(* CoDeSys 2.3.9.35 project: Program stor plattform.pro *)
(* Libraries: Standard.lib 2.12.10 13:48:34, Iecsfc.lib 2.12.10 13:48:34, SYSLIBCALLBACK.LIB 2.12.10 13:48:34 *)

(* PLC configuration (modules and I/O channels)
K-Bus [K_Bus] node 0, in %IB0 out %QB0
DIN1 AT %IX2300.0 [BOOLOnX_I] Internal Digital Input Bit 1
DIN2 AT %IX2300.1 [BOOLOnX_I] Internal Digital Input Bit 2
DOUT1 AT %QX2300.0 [BOOLOnX_Q] Internal Digital Output Bit 1
DOUT2 AT %QX2300.1 [BOOLOnX_Q] Internal Digital Output Bit 2
Fieldbus variables [FB_VARS] node 3, in %IB0 out %QB0
Flag variables [FLAG_VARS] node 4, in %IB0 out %QB0
*)

(* Task configuration *)
TASK NewTask (PRIORITY := 15); (* freewheeling *)
	PLC_PRG();
	Read_Pos();
	Read_Param();
	SET_STEP();
END_TASK

(* Global variable list: Global_Variables *)
VAR_GLOBAL
	(*Manual mode variabler*)
	STOP: BOOL;
	JOGM1: BOOL;
	JOGP1: BOOL;
	JOGM2: BOOL;
	JOGP2: BOOL;
	JOGM3: BOOL;
	JOGP3: BOOL;
	GO_UP: BOOL;
	GO_DOWN: BOOL;
	GO_HOME: BOOL;
	Manual_speed: INT:=300;

	(*Motor 1*)
	M1_Cont_inhibit AT%QX2404.8 : BOOL;
	DATA_IN_M1: INT;
	Y_M1: INT;
	M1_ANGLE: REAL;

	(*Motor 2*)
	M2_Cont_inhibit AT%QX2411.8 : BOOL;
	DATA_IN_M2: INT;
	Y_M2: INT;
	M2_ANGLE:REAL;

	(*Motor 3*)
	M3_Cont_inhibit AT%QX2418.8 : BOOL;
	DATA_IN_M3: INT;
	Y_M3: INT;
	M3_ANGLE:REAL;




   (*MOTOR 1 Set Points*)
	p1_step: INT;
	(*MOTOR 2 Set Points*)
	p2_step: INT;
	(*MOTOR 3 Set points*)
	p3_step: INT;


	(*Platform angle Set Points*)
	pitch:REAL;
	roll:REAL;


	(*MODES*)
	ENABLE: BOOL;  (*Enables the Drives*)
	manual_run: BOOL;		(* Set specified position *)
	wave_run: BOOL; 	(* Wave PROGRAM *)
	input_run: BOOL;		(* Roll / Pitch input from other sources *)

	SIMULATION_UDP: BOOL;

	LOGG :BOOL;

END_VAR

VAR_GLOBAL CONSTANT

	l1:INT:=150;  			(*lower arm in mm*)
	l2:INT:=330;  			(*upper arm in mm*)
	l3:INT:=1075; 			(*length between joints p1, p2, p3*)
	l4:INT:=931;			(*length of platform center from p1*)
	l5:INT := 311;
	l6:INT := 620;
	mid_length:INT:=370;	(*mid length of both arms combined*)
	min_angle:INT:= -125;
	max_angle:INT:= 0;
	max_roll:INT:=10;
	min_roll:INT:=-10;
	max_pitch:INT:=10;
	min_pitch: INT:=-10;
	am:REAL:=57.2958; 			(*arcminute constant*)

END_VAR

(* POU PLC_PRG, ST *)
PROGRAM PLC_PRG
VAR
	RPTS: ROLL_PITCH_TO_STEP;
	Read_par: BOOL;

END_VAR
(* PROGRAM VELGER. *)

IF(wave_run) AND NOT(input_run) AND NOT(manual_run) THEN
WAVE_V3();
END_IF;

IF(input_run) AND NOT(wave_run) AND NOT(manual_run) THEN
INPUT_MODE();
END_IF;

IF(manual_run) AND NOT(input_run) AND NOT(wave_run) THEN
MANUAL();
END_IF;

(*Setter Plattformen i 0 pos.*)
IF( NOT wave_run AND NOT input_run AND NOT manual_run) THEN
RPTS(roll_angle:=0,pitch_angle:=0);
p1_step:=RPTS.step1;
p2_step:=RPTS.step2;
p3_step:=RPTS.step3;
END_IF;
END_PROGRAM

(* POU Calculations/ROLL_PITCH_TO_STEP, ST *)
FUNCTION_BLOCK ROLL_PITCH_TO_STEP (*ROLL PITCH CALCULATOR*)
VAR_INPUT
	roll_angle:REAL;
	pitch_angle:REAL;
END_VAR
VAR_OUTPUT
	step1: INT;
	step2: INT;
	step3: INT;
END_VAR
VAR
	a: REAL;
	b: REAL;
	mid_length1: REAL;
	c: REAL;
	HTS1:HIGHT_TO_STEP;
	HTS2:HIGHT_TO_STEP;
	HTS3:HIGHT_TO_STEP;
	set_p1:INT;
	set_p2:INT;
	set_p3:INT;
END_VAR
IF(roll_angle >= max_roll) THEN
roll_angle:=max_roll;
ELSIF(roll_angle <= min_roll) THEN
roll_angle:=min_roll;
END_IF;

IF(pitch_angle >=max_pitch) THEN
pitch_angle:= max_pitch;
ELSIF(pitch_angle <= min_pitch) THEN
pitch_angle:=min_pitch;
END_IF

b:=(SIN(pitch_angle/am));

set_p1:= REAL_TO_INT(mid_length+b*l6);
mid_length1:=mid_length-b*l5;

a:=(SIN(roll_angle/am)*l3)/2;
set_p2:= REAL_TO_INT(mid_length1-a);
set_p3:= REAL_TO_INT(mid_length1+a);

HTS1(length:=set_p1);
HTS2(length:=set_p2);
HTS3(length:=set_p3);
step1:=HTS1.step;
step2:=HTS2.step;
step3:=HTS3.step;
END_FUNCTION_BLOCK

(* POU Calculations/HIGHT_TO_STEP, ST *)
FUNCTION_BLOCK HIGHT_TO_STEP
VAR_INPUT
	length:INT;
END_VAR
VAR_OUTPUT
	angle:REAL;
	step:INT;
END_VAR
VAR
	b: REAL;
	a: REAL;
	c: REAL;
	h: INT;
END_VAR
h:=length;
IF(h > 480) THEN
h:=480;
END_IF
IF(h < 260) THEN
h:=260;
END_IF

a:=(l1*l1)+(h*h)-(l2*l2);
b:=(2*l1*h);
angle:=-60*ACOS(a/b)+125;
step:= REAL_TO_INT((14000/125)*angle+2000);
END_FUNCTION_BLOCK

(* POU Progamer/WAVE_V3, ST *)
PROGRAM WAVE_V3
VAR
	X_M1 :REAL;
	X_M2: REAL := -1.5;
	X_M3: REAL := 1.5;
	top_M1: BOOL;
	top_M2: BOOL;
	top_M3: BOOL;
	Speed1 : REAL := 0.1;
	Speed2 : REAL := 0.1;
	Speed3 : REAL := 0.1;
	HTS1: HIGHT_TO_STEP;
	HTS2: HIGHT_TO_STEP;
	HTS3: HIGHT_TO_STEP;

	Ampl: INT := 30;
END_VAR
(* SINUS WAWE M1*)
IF (X_M1 <= 1.57) AND NOT(top_M1) THEN
X_M1 := (X_M1 + Speed1);
END_IF

IF (X_M1 >= 1.57) THEN
top_M1 := TRUE;
END_IF

IF top_M1 THEN
X_M1 := (X_M1 - Speed1);
END_IF

IF (X_M1 <= -1.57) THEN
top_M1 := FALSE;
END_IF
(*
HTS1(length:= 370 + REAL_TO_INT(110 * SIN (X_M1)));*)

HTS1(length:= 370 + REAL_TO_INT(Ampl * SIN (X_M1)));

(* SINUS WAWE M2*)
IF (X_M2 <= 1.57) AND NOT(top_M2) THEN
X_M2 := (X_M2 + Speed2);
END_IF

IF (X_M2 >= 1.57) THEN
top_M2 := TRUE;
END_IF

IF top_M2 THEN
X_M2 := (X_M2 - Speed2);
END_IF

IF (X_M2 <= -1.57) THEN
top_M2 := FALSE;
END_IF

HTS2 (length:= 370 + REAL_TO_INT(Ampl * SIN (X_M2)));


(* SINUS WAWE M3*)

IF (X_M3 <= 1.57) AND NOT(top_M3) THEN
X_M3 := (X_M3 + Speed3);
END_IF

IF (X_M3 >= 1.57) THEN
top_M3 := TRUE;
END_IF

IF top_M3 THEN
X_M3 := (X_M3 - Speed3);
END_IF

IF (X_M3 <= -1.57) THEN
top_M3 := FALSE;
END_IF

HTS3 (length:= 370 + REAL_TO_INT(Ampl * SIN (X_M3)));




p1_step:= HTS1.step;
p2_step:= HTS2.step;
p3_step:= HTS3.step;
M1_ANGLE:=HTS1.angle;
M2_ANGLE:=HTS2.angle;
M3_ANGLE:=HTS3.angle;
END_PROGRAM

(* POU Progamer/INPUT_MODE, ST *)
PROGRAM INPUT_MODE
VAR

    (* Verdier hentet fra UDP stream *)
	Input_Roll: WORD;
	Input_Pitch: WORD;
	sim_roll: REAL;
	sim_pitch: REAL;
	INPUT_roll_real: REAL;
	INPUT_pitch_real: REAL;
	rpts: ROLL_PITCH_TO_STEP;

	pitch_real: INT;
	roll_real: INT;
	roll_old: REAL:=0;
	pitch_old: REAL:=0;
	roll_new: REAL;
	pitch_new: REAL;
	roll_new_int: INT;
	pitch_new_int: INT;
END_VAR
roll_new_int :=WORD_TO_INT(Input_Roll);
pitch_new_int:=WORD_TO_INT(Input_Pitch);

roll_new:=2*INT_TO_REAL(-roll_new_int) / 1000;
pitch_new:=2*INT_TO_REAL(pitch_new_int) / 1000;

INPUT_roll_real:=(roll_new*0.1+roll_old*0.9);
INPUT_pitch_real:=(pitch_new*0.1+pitch_old*0.9);
IF SIMULATION_UDP THEN
INPUT_roll_real := sim_roll;
INPUT_pitch_real := sim_pitch;
END_IF
rpts(roll_angle:=INPUT_ROLL_REAL,pitch_angle:=INPUT_PITCH_REAL);

p1_step:=rpts.step1;
p2_step:=rpts.step2;
p3_step:=rpts.step3;

roll_old:=INPUT_roll_real;
pitch_old:=INPUT_pitch_real;
END_PROGRAM

(* POU Progamer/MANUAL, ST *)
PROGRAM MANUAL
VAR
	Speed : INT := 200;
END_VAR
(* Begrenser verdien til pX_step *)
IF p1_step > 14000 THEN p1_step := 14000; END_IF
IF p2_step > 14000 THEN p2_step := 14000; END_IF
IF p3_step > 14000 THEN p3_step := 14000; END_IF

IF p1_step < 2000 THEN p1_step := 2000; END_IF
IF p2_step < 2000 THEN p2_step := 2000; END_IF
IF p3_step < 2000 THEN p3_step := 2000; END_IF

(* Motor1 opp *)
IF JOGP1 THEN
p1_step := p1_step+Speed;
END_IF

(* Motor1 ned *)
IF JOGM1 THEN
p1_step := p1_step-Speed;
END_IF

(* Motor2 opp *)
IF JOGP2 THEN
p2_step := p2_step+Speed;
END_IF

(* Motor2 ned *)
IF JOGM2 THEN
p2_step := p2_step-Speed;
END_IF

(* Motor3 opp *)
IF JOGP3 THEN
p3_step := p3_step+Speed;
END_IF

(* Motor3 Ned *)
IF JOGM3 THEN
p3_step := p3_step-Speed;
END_IF

(*Kjører alle motorene opp *)
IF GO_UP THEN
p1_step := p1_step+Speed;
p2_step := p2_step+Speed;
p3_step := p3_step+Speed;
END_IF

(*Kjører alle motorene ned *)
IF GO_DOWN THEN
p1_step := p1_step-Speed;
p2_step := p2_step-Speed;
p3_step := p3_step-Speed;
END_IF
END_PROGRAM

(* POU Read Values/Read_Pos, ST *)
PROGRAM Read_Pos
VAR_INPUT
END_VAR
VAR
(*Motor 1*)
	In_data_1 AT %IW2405: WORD;
	In_data_2 AT %IW2406: WORD;
	Data_in_m1_temp: WORD;
(*Motor 2*)
	In_data_3  AT %IW2412: WORD;
	In_data_4 AT %IW2413: WORD;
	Data_in_m2_temp: WORD;
(*Motor 3*)
	In_data_5 AT %IW2419: WORD;
	In_data_6 AT %IW2420: WORD;
	data_in_m3_temp: WORD;
	CA: CALCULATED_ACTUALS;
	roll_actual: WORD;
	pitch_actual: WORD;
	PA: REAL;
	PR: REAL;


(* SEND TO JAVA *)
	STH1: STEP_TO_HIGHT;
	STH2: STEP_TO_HIGHT;
	STH3: STEP_TO_HIGHT;


	h1 : INT;
	h2 : INT;
	h3 : INT;
	h4:INT;
	Z : INT;
	Zo AT %MW1: INT;

	hm1: INT;
	hm2: INT;
	hm3: INT;
END_VAR
(*Leser av posisjonsdata til motor 1*)
Data_in_m1_temp:= ROL(In_data_1 + In_data_2, 8);
DATA_IN_M1 := WORD_TO_INT(Data_in_m1_temp);

(*Leser av posisjonsdata til motor 2*)
Data_in_m2_temp := ROL(In_data_3 + In_data_4, 8);
DATA_IN_M2 := WORD_TO_INT(Data_in_m2_temp);

(*Leser av posisjonsdata til motor 3*)
data_in_m3_temp := ROL(In_data_5 + In_data_6, 8);
DATA_IN_M3 := WORD_TO_INT(Data_in_m3_temp);
ca();

PA := (CA.a_pitch);
PR := (CA.a_roll);

roll_actual := REAL_TO_INT(PR*1000);
pitch_actual := REAL_TO_INT(PA*1000);
(*
STH1(stepp:=DATA_IN_M1);
STH2(stepp:=DATA_IN_M2);
STH3(stepp:=DATA_IN_M3);
*)

STH1(stepp:=p1_step);
STH2(stepp:=p2_step);
STH3(stepp:=p3_step);


h1 := STH1.h;
h2 := STH2.h;
h3 := STH3.h;

hm1 := h1 - 416;
hm2 := h2 - 416;
hm3 := h3 - 416;

h4 := (h2+h3)/2;

Z := h1 - (h1-h4)/3;


Zo := Z - 416 +10000;
END_PROGRAM

(* POU Calculations/CALCULATED_ACTUALS, ST *)
FUNCTION_BLOCK CALCULATED_ACTUALS
(*Uses step reading from encoders to calculate hight and angle on each motor, pitch and roll*)
VAR_INPUT
END_VAR
VAR_OUTPUT
	a_hight1: INT;
	a_hight2: INT;
	a_hight3: INT;
	a_angle1: REAL;
	a_angle2: REAL;
	a_angle3: REAL;
	a_roll:	  REAL;
	a_pitch:  REAL;
	a_roll_1 AT %MW10:	INT;
	a_pitch_1 AT %MW15:  INT;

END_VAR
VAR
	st1: STEP_TO_HIGHT;
	st2: STEP_TO_HIGHT;
	st3: STEP_TO_HIGHT;
	a: REAL;
	b: REAL;
	c: REAL;
	d: REAL;
END_VAR
st1(stepp:=(DATA_IN_M1));
st2(stepp:=(DATA_IN_M2));
st3(stepp:=(DATA_IN_M3));

a_hight1:=st1.h;
a_hight2:=st2.h;
a_hight3:=st3.h;
a_angle1:=st1.a;
a_angle2:=st2.a;
a_angle3:=st3.a;

a:=(a_hight3-a_hight2);
b:=(a/l3);
a_roll:=am*ASIN(b);


c:=(a_hight2+a_hight3)/2;
d:=(a_hight1-c)/l4;
a_pitch:=am*ASIN(d);


a_roll_1 := REAL_TO_INT(a_roll*100) + 10000;
a_pitch_1 := REAL_TO_INT(a_pitch*100) + 10000;
END_FUNCTION_BLOCK

(* POU Calculations/STEP_TO_HIGHT, ST *)
FUNCTION_BLOCK STEP_TO_HIGHT
VAR_INPUT
(* Antall steg *)
	stepp: INT;

END_VAR
VAR_OUTPUT
(* Høyde fra aksling motor til senter kule på plattform *)
	h: INT;
	a: REAL; (* VINKEL *)
END_VAR
VAR
	b: REAL;
	a1: REAL;
END_VAR
b:=INT_TO_REAL(stepp);
a:=(b/(14000))*120-120;
a1 := a/am;
h:=REAL_TO_INT(l1*COS(a1)+SQRT(l2*l2-l1*l1*SIN(a1)*SIN(a1)));
END_FUNCTION_BLOCK

(* POU Read Values/Read_Param, ST *)
PROGRAM Read_Param
VAR

	Management: WORD;
	Word0 AT %QW2400: WORD;
	Word1 AT %QW2401: WORD;
	Read_value0 AT %IW2400: WORD;
	Read_value1 AT %IW2401: WORD;
	Out_put0: WORD;
	Out_put1: WORD;
	Out: INT;
	Data_Out: INT;
	Read_par: BOOL;
	Par_nr:INT;
END_VAR
IF(Read_par) THEN
Management := INT_TO_WORD(1 + 16 + 32 + 64);
Word0 := ROR(Management , 8);

Par_nr := INT_TO_WORD(8398);
Word1 := ROR(Par_nr, 8);

Out_put0 := ROL(Read_value0 , 8);
Out_put1 := ROL(Read_value1 , 8);

Data_Out := WORD_TO_INT( Read_value0 + Read_value1);

ELSE
Management := INT_TO_WORD(1 + 16 + 32);
Word0 := ROR(Management , 8);
END_IF
END_PROGRAM

(* POU SET_STEP, ST *)
PROGRAM SET_STEP
VAR
	SET_M1:DINT;
	STEP_M1: INT;
	SET_M2:DINT;
	STEP_M2: INT;
	SET_M3:DINT;
	STEP_M3: INT;
END_VAR
(* P1-3_STEP globale variabler for ønsket Steg *)
(* DATA_IN_M1-M3 steg verdier avlest fra profibus *)
(*M1*)
IF(DATA_IN_M1 > P1_STEP) THEN
(*ned*)
STEP_M1:=REAL_TO_INT((P1_STEP-DATA_IN_M1)/3);
IF(STEP_M1 < -2000) THEN
STEP_M1:= -2000;
END_IF;
(*OPP*)
ELSIF(DATA_IN_M1 < P1_STEP) THEN
STEP_M1:=REAL_TO_INT((P1_STEP - DATA_IN_M1)/3);
IF(STEP_M1 > 2000) THEN
STEP_M1:=2000;
END_IF;
ELSE
STEP_M1:=0;
END_IF;
M1(SPEED_DIR:=STEP_M1);


(*M2*)
IF(DATA_IN_M2 > P2_STEP) THEN
(*NED*)
STEP_M2:=REAL_TO_INT((P2_STEP-DATA_IN_M2)/3);
IF(STEP_M2 < -2000) THEN
STEP_M2:= -2000;
END_IF;
(*OPP*)
ELSIF(DATA_IN_M2 < P2_STEP) THEN
STEP_M2:=REAL_TO_INT((P2_STEP - DATA_IN_M2)/3);
IF(STEP_M2 > 2000) THEN
STEP_M2:=2000;
END_IF;
ELSE
STEP_M2:=0;
END_IF;
M2(SPEED_DIR:=STEP_M2);

(*M3*)
IF(DATA_IN_M3 > P3_STEP) THEN
STEP_M3:=REAL_TO_INT((P3_STEP-DATA_IN_M3)/3);
IF(STEP_M3 < -2000) THEN
STEP_M3:= -2000;
END_IF;
ELSIF(DATA_IN_M3 < P3_STEP) THEN
STEP_M3:=REAL_TO_INT((P3_STEP - DATA_IN_M3)/3);
IF(STEP_M3 < -2000) THEN
STEP_M3:=-2000;
END_IF;
ELSE
STEP_M3:=0;
END_IF;
M3(SPEED_DIR:=STEP_M3);
END_PROGRAM

(* POU RUN Motor/M1, ST *)
FUNCTION M1 : BOOL
VAR_INPUT
	SPEED_DIR:INT;
END_VAR
VAR
	P0_1_M1 AT %QW2404: WORD;
	P0_2_M1 AT %QW2405: WORD;
END_VAR
IF (ENABLE) THEN
P0_1_M1 := ROR(INT_TO_WORD( 2 + 4),8);	(*Enable signal til M1 sent på ORD 1*)
P0_2_M1 := ROR(INT_TO_WORD(SPEED_DIR), 8);	(* Setter hastigheten til M1 på ord 2 *)
ELSE
M1_Cont_inhibit := TRUE;
END_IF
END_FUNCTION

(* POU RUN Motor/M2, ST *)
FUNCTION M2 : BOOL
VAR_INPUT
	SPEED_DIR:INT;
END_VAR
VAR
	P0_1_M2 AT %QW2411: WORD;
	P0_2_M2 AT %QW2412: WORD;
END_VAR
IF (ENABLE) THEN
P0_1_M2 := ROR(INT_TO_WORD( 2 + 4), 8);		(*Enable signal til M2 sent på ORD 1*)
P0_2_M2 := ROR(INT_TO_WORD(SPEED_DIR), 8);	(* Setter hastigheten til M2 på ord 2 *)
ELSE
M2_Cont_inhibit := TRUE;
END_IF
END_FUNCTION

(* POU RUN Motor/M3, ST *)
FUNCTION M3 : BOOL
VAR_INPUT
	SPEED_DIR:INT;
END_VAR
VAR
	P0_1_M3 AT %QW2418: WORD;
	P0_2_M3 AT %QW2419: WORD;
END_VAR
IF (ENABLE) THEN
P0_1_M3 := ROR(INT_TO_WORD( 2 + 4), 8);		(*Enable signal til M3 sent på ord 1*)
P0_2_M3 := ROR(INT_TO_WORD(Speed_DIR), 8);	(* Setter hastigheten til M3 på ord 2 *)
ELSE
M3_Cont_inhibit := TRUE;
END_IF
END_FUNCTION

(* Visualisation Graph
rectangle at (680,40)-(851,151): text "record"; alarm colour if .LOGG; toggles .LOGG
3 elements of other kinds (tables, trends, ...) not read
*)

(* Visualisation HOME
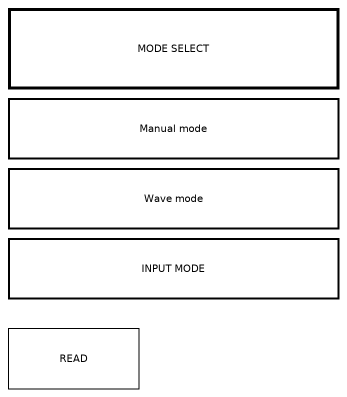
rectangle at (10,10)-(341,91): text "MODE SELECT"
rectangle at (10,100)-(341,161): text "Manual mode"; alarm colour if .manuell_styring; opens Manual_mode
rectangle at (10,170)-(341,231): text "Wave mode"; alarm colour if .wave_pattern; opens Wave_mode
rectangle at (10,240)-(341,301): text "INPUT MODE"; alarm colour if .Udp_Stream_mode; opens UDP
rectangle at (10,330)-(141,391): text "READ"; taps Read_Param.Read_par
*)

(* Visualisation Manual_mode
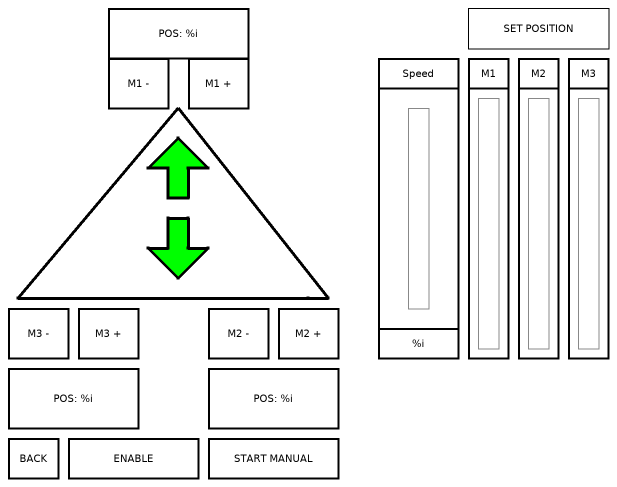
rectangle at (190,50)-(251,101): text "M1 +"; alarm colour if .JOGP; taps JOGP1
rectangle at (110,50)-(171,101): text "M1 -"; alarm colour if .JOGM; taps JOGM1
rectangle at (80,300)-(141,351): text "M3 +"; alarm colour if .JOGP; taps JOGP3
rectangle at (280,300)-(341,351): text "M2 +"; alarm colour if .JOGP; taps JOGP2
rectangle at (10,300)-(71,351): text "M3 -"; alarm colour if .JOGM; taps JOGM3
rectangle at (210,300)-(271,351): text "M2 -"; alarm colour if .JOGM; taps JOGM2
rectangle at (110,0)-(251,51): text "POS: %i"; shows .DATA_IN_M1
rectangle at (210,360)-(341,421): text "POS: %i"; shows .DATA_IN_M2
rectangle at (10,360)-(141,421): text "POS: %i"; shows .DATA_IN_M3
polygon at (150,130)-(210,190): taps .GO_UP
polygon at (150,210)-(210,270): taps .GO_DOWN
rectangle at (210,430)-(341,471): text "START MANUAL"; alarm colour if .manual_run; toggles manual_run
rectangle at (70,430)-(201,471): text "ENABLE"; alarm colour if .ENABLE; toggles .ENABLE
rectangle at (380,50)-(461,81): text "Speed"
rectangle at (380,320)-(461,351): text "%i"; shows .Manual_speed
rectangle at (10,430)-(61,471): text "BACK"; opens HOME
rectangle at (470,50)-(511,81): text "M1"
rectangle at (520,50)-(561,81): text "M2"
rectangle at (570,50)-(611,81): text "M3"
rectangle at (470,0)-(611,41): text "SET POSITION"
9 more shapes without text or variables
*)

(* Visualisation UDP
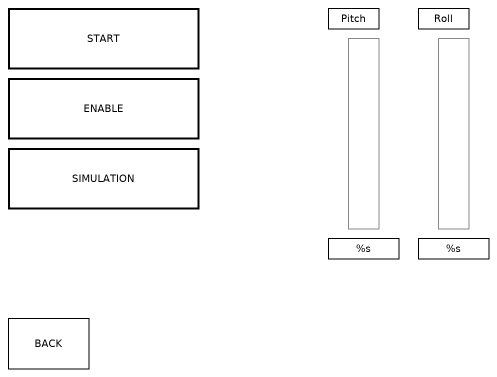
rectangle at (10,10)-(201,71): text "START"; alarm colour if .INPUT_RUN; toggles .input_run
rectangle at (10,80)-(201,141): text "ENABLE"; alarm colour if .ENABLE; toggles .ENABLE
rectangle at (10,320)-(91,371): text "BACK"; opens HOME; runs HOME
rectangle at (330,10)-(381,31): text "Pitch"
rectangle at (420,10)-(471,31): text "Roll"
rectangle at (330,240)-(401,261): text "%s"; shows INPUT_MODE.sim_pitch
rectangle at (420,240)-(491,261): text "%s"; shows INPUT_MODE.sim_roll
rectangle at (10,150)-(201,211): text "SIMULATION"; alarm colour if .SIMULATION_UDP; toggles .SIMULATION_UDP
2 more shapes without text or variables
*)

(* Visualisation Wave_mode
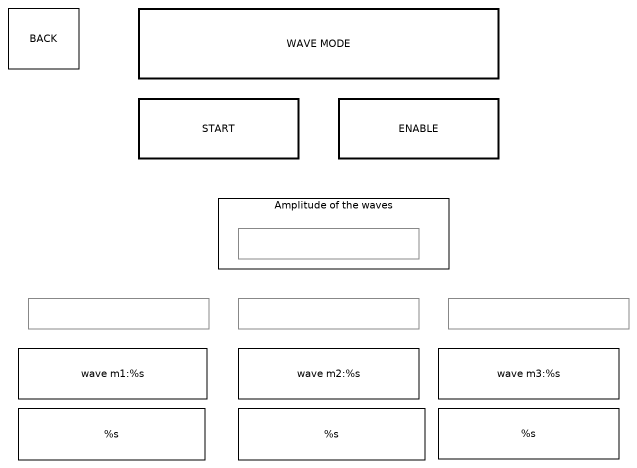
rectangle at (220,210)-(451,281): text "Amplitude of the waves"
rectangle at (20,420)-(207,472): text "%s"; shows .DATA_IN_M1
rectangle at (20,360)-(209,411): text "wave m1:%s"; shows .p1_step
rectangle at (240,420)-(427,472): text "%s"; shows .DATA_IN_M2
rectangle at (440,420)-(621,471): text "%s"; shows .DATA_IN_M3
rectangle at (240,360)-(421,411): text "wave m2:%s"; shows .p2_step
rectangle at (440,360)-(621,411): text "wave m3:%s"; shows .p3_step
rectangle at (340,110)-(501,171): text "ENABLE"; alarm colour if .ENABLE; toggles .ENABLE
rectangle at (140,20)-(501,91): text "WAVE MODE"; alarm colour if .wave_pattern
rectangle at (140,110)-(301,171): text "START"; alarm colour if .wave_run; toggles .wave_run
rectangle at (10,20)-(81,81): text "BACK"; opens HOME
4 more shapes without text or variables
*)
